{attribute 'qualified_only'}
VAR_GLOBAL
	bStartLight : BOOL;
	bStopLight : BOOL;
	eCraneMode : E_CraneMode;
	eCraneStatus : E_CraneStatus;
	fNormalizedOutput : LREAL;
END_VAR

(* stored: Version 1.1.0.1, ProductVersion 3.1.4024.10
   GVL Outputs: Id {04c7e31d-42dd-42ce-9d57-ed88c639b70d} *)
